{attribute 'GeneratedUsingTerminal: EK1122-0000-0018'}
{attribute addProperty BoxType "EK1122-0000-0018"}
{attribute addProperty Id "Beckhoff_EPP6xxxsub_EK1100EK1100_AB5A94672A_0001_EPP6001_0002_0016EPP6001_B965E9F560A_0002_EPP6001_0002_0017EPP6001_B965E9F560A_0003_EPP6001_0002_0018EPP6001_B965E9F560A_0004_EPP6002_0002_0016EPP6002_EA7A2404108A_0005_EPP6002_0002_0017EPP6002_EA7A2404108A_0006_EPP6002_0002_0018EPP6002_EECF1379108A_0007_EPP6002_0002_0019EPP6002_EECF1379108A_0008_EPP6090_0000_0017EPP6090_1BDB3CCC22A_0009_EPP6228_0022_0016EPP6228_0C20E27E36"}
{attribute addProperty CRC "2464416817"}
{attribute addProperty Size "672"}
TYPE Beckhoff_EPP6xxxEK1122_92E40431 EXTENDS EK1122_AB5A9467 :
STRUCT
	{attribute addProperty Name "Beckhoff_EPP6xxxsub_EK1100"}
	Beckhoff_EPP6xxxsub_EK1100 : EK1100_AB5A9467;
	{attribute addProperty Name "A_0001_EPP6001_0002_0016"}
	A_0001_EPP6001_0002_0016 : EPP6001_B965E9F5;
	{attribute addProperty Name "A_0002_EPP6001_0002_0017"}
	A_0002_EPP6001_0002_0017 : EPP6001_B965E9F5;
	{attribute addProperty Name "A_0003_EPP6001_0002_0018"}
	A_0003_EPP6001_0002_0018 : EPP6001_B965E9F5;
	{attribute addProperty Name "A_0004_EPP6002_0002_0016"}
	A_0004_EPP6002_0002_0016 : EPP6002_EA7A2404;
	{attribute addProperty Name "A_0005_EPP6002_0002_0017"}
	A_0005_EPP6002_0002_0017 : EPP6002_EA7A2404;
	{attribute addProperty Name "A_0006_EPP6002_0002_0018"}
	A_0006_EPP6002_0002_0018 : EPP6002_EECF1379;
	{attribute addProperty Name "A_0007_EPP6002_0002_0019"}
	A_0007_EPP6002_0002_0019 : EPP6002_EECF1379;
	{attribute addProperty Name "A_0008_EPP6090_0000_0017"}
	A_0008_EPP6090_0000_0017 : EPP6090_1BDB3CCC;
	{attribute addProperty Name "A_0009_EPP6228_0022_0016"}
	A_0009_EPP6228_0022_0016 : EPP6228_0C20E27E;
END_STRUCT
END_TYPE

(* stored: Version 1.2.0.0, ProductVersion 3.1.4024.9
   DUT Beckhoff_EPP6xxxEK1122_92E40431: Id {2335c5e8-a259-4fa7-ac21-65805e60f2af} *)
